FUNCTION_BLOCK FB_Syntax_IfMultilineCalls
VAR
    sStr1   : STRING(80);
    sStr2   : STRING(80);
    sResult : STRING(255);
    rTarget : REFERENCE TO INT;
    nVal    : INT;
    bOk     : BOOL;
END_VAR

IF len(sStr1) > 0 AND len(sStr2) > 0 THEN
    bOk := FALSE;
ELSE
    bOk := TRUE;
END_IF

IF NOT __ISVALIDREF(rTarget) THEN
    nVal := 0;
ELSE
    nVal := rTarget;
END_IF

IF (len(sStr1) > 0) AND (len(sStr2) > 0) AND (len(sResult) = 0) THEN
    bOk := TRUE;
END_IF

END_FUNCTION_BLOCK

(* stored: Version 1.1.0.1, ProductVersion 3.1.4024.16
   POU FB_Syntax_IfMultilineCalls: Id {5b203008-c657-4a7f-a331-701f05bebd84}, SpecialFunc None *)
